{attribute 'GeneratedUsingTerminal: EK1100-0000-0018'}
{attribute addProperty BoxType "EK1100-0000-0018"}
{attribute addProperty Id "Beckhoff_EQ1xxxEK1122Beckhoff_EQ1xxxEK1122_E78E0C9478"}
{attribute addProperty CRC "4135334461"}
{attribute addProperty Size "78"}
TYPE Beckhoff_EQ1xxx_F67C323D EXTENDS EK1100_1FC0878B :
STRUCT
	{attribute addProperty Name "Beckhoff EQ1xxxEK1122"}
	{attribute addProperty PreviousPort "Beckhoff EQ1xxx : B"}
	Beckhoff_EQ1xxxEK1122 : Beckhoff_EQ1xxxEK1122_E78E0C94;
END_STRUCT
END_TYPE

(* stored: Version 1.2.0.0, ProductVersion 3.1.4024.9
   DUT Beckhoff_EQ1xxx_F67C323D: Id {85702d5d-8a30-4df0-8c6f-0351c350e471} *)
